FUNCTION_BLOCK AX_FB_SR_T_FF (* Realizes a bistable set-dominat latch plus Toggle *)
  (* Standard: 61499-1; Description: Copyright (c) 2023 Martin Erich Jobst This program and the accompanying materials are made available under the terms of the Eclipse Public License 2.0 which is available at https://www.eclipse.org/legal/epl-2.0/ SPDX-License-Identifier: EPL-2.0 *)
  (* Version 3.0, 2025-04-14, Patrick Aigner, changed package *)
  (* Version 1.0, 2023-04-28, Martin Jobst *)
  PACKAGE adapter::bistableElements;
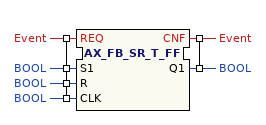
  EVENT_INPUT
    REQ WITH S1, R, CLK; (* Normal Execution Request *)
  END_EVENT
  EVENT_OUTPUT
    CNF WITH Q1; (* Execution Confirmation *)
  END_EVENT
  VAR_INPUT
    S1 : BOOL; (* Set *)
    R : BOOL; (* Reset *)
    CLK : BOOL; (* Clock *)
  END_VAR
  VAR_OUTPUT
    Q1 : BOOL; (* Output *)
  END_VAR
  VAR
    EDGE : BOOL := TRUE;
  END_VAR
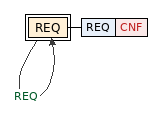
  EC_STATES
    REQ : REQ -> CNF;
  END_STATES
  EC_TRANSITIONS
    REQ TO REQ := REQ;
  END_TRANSITIONS
  ALGORITHM REQ IN ST:
IF S1 THEN
	Q1 := BOOL#TRUE;
ELSIF R THEN
	Q1 := BOOL#FALSE;
ELSIF CLK AND NOT EDGE THEN
	Q1 := NOT Q1;
END_IF;
EDGE := NOT CLK;
  END_ALGORITHM
END_FUNCTION_BLOCK
